PROGRAM PRG_TCPIP 
VAR	
	bInit 						:BOOL := TRUE;
	bReset						:BOOL;
	
	stReadTCP					:ST_TCPConnection;
	fbReadFromCameraTCP			:FB_ReadTCP;
	bConnectToReadSocket		:BOOL;
	
	stWriteTCP					:ST_TCPConnection;
	fbWriteToHLZ				:FB_WriteTCP;
	bConnectToWriteSocket		:BOOL;
END_VAR

//Init
IF bInit THEN	
	bInit := FALSE;
END_IF


A_ReadFromCamera();
A_WriteToHlz();


//Reset Commands
GVL_HMI.stTCPConnectionCmd.bResetRegistry := FALSE;


IF GVL_HMI.stTCPConnectionCmd.bWriteSocketConnect THEN
	GVL_HMI.stTCPConnectionCmd.bReadSocketConnect := FALSE;
	
ELSIF GVL_HMI.stTCPConnectionCmd.bReadSocketConnect THEN
	GVL_HMI.stTCPConnectionCmd.bWriteSocketConnect := FALSE;
END_IF;

ACTION A_ReadFromCamera:
//Initialize Read TCP
stReadTCP.sRemoteHost := '10.12.5.10';
stReadTCP.nRemotePort := 51236;
stReadTCP.tTimeOut := T#45S;
stReadTCP.bSocketConnect := GVL_HMI.stTCPConnectionCmd.bReadSocketConnect;
stReadTCP.bReset := GVL_HMI.stTCPConnectionCmd.bResetRegistry;

//Call Read TCP
fbReadFromCameraTCP(
	stTCPConnection:=stReadTCP,
	aEANRegistry=>GVL_HMI.stTCPConnectionStatus.aEANRegistry,
	bIsConnected=>GVL_HMI.stTCPConnectionStatus.bCameraReadSocketIsConnected);
END_ACTION

ACTION A_WriteToHlz:
//Initialize Write TCP
stWriteTCP.sRemoteHost := '10.12.5.10';
stWriteTCP.nRemotePort := 51237;
stWriteTCP.tTimeOut := T#45S;
stWriteTCP.bSocketConnect := GVL_HMI.stTCPConnectionCmd.bWriteSocketConnect;
stWriteTCP.bReset := GVL_HMI.stTCPConnectionCmd.bResetRegistry;


//Call Write TCP
fbWriteToHLZ(
	aEANRegistry:=fbReadFromCameraTCP.aEANRegistry,
	stTCPConnection:=stWriteTCP,
	bIsConnected=>GVL_HMI.stTCPConnectionStatus.bHlzWriteSocketIsConnected);
END_ACTION

END_PROGRAM

(* stored: Version 1.1.0.1, ProductVersion 3.1.4024.12
   POU PRG_TCPIP: Id {e26f0609-c5dd-4c0e-bab1-8c4ef3547268}, SpecialFunc None
   Action A_ReadFromCamera: Id {fa2fa6f9-072d-42cf-9835-c8d01007dda3}
   Action A_WriteToHlz: Id {029a87b5-d519-4d88-b685-d7af7eb27bad} *)
